TYPE "ValveAlr"
VERSION : 0.1
// Block: ValveAlr
   STRUCT
      TimeOutRest : Bool;
      TimeOutWork : Bool;
      LimitSwitches : Bool;
   END_STRUCT;

END_TYPE
